TYPE DUT_ST_InfoData :
STRUCT
	// Safety Groups use this structure
	usiMapState 			: 	USINT ;
	usiMapDiag  			: 	USINT ;
END_STRUCT
END_TYPE

(* stored: Version 1.1.0.1, ProductVersion 3.1.0.18
   DUT DUT_ST_InfoData: Id {e5b62de3-a32e-4f0f-aa87-2ced50560f64} *)
